(* IEC 61131-3 sources: tutorials/projects/ch05-2/PROGRAM, 4 files *)

(* ---- types.st ---- *)
(* 有初始化的数据类型 *)
TYPE BYTE_WITH_RANGE :
    SINT := 16#1A; (* 初始化为 0x1A *)
END_TYPE

(** 数组数据类型 *)
TYPE ARRAY_BYTES_WITH_RANGE :
    ARRAY [0..3] OF BYTE_WITH_RANGE;
END_TYPE

(* 枚举类型的数据类型: 机器状态 *)
TYPE ENUM_STATE_MACHINE : (
        INIT,
        PREPARING,
        RUNNING,
        STOPPED
    ) ;
END_TYPE

(*结构化的数据类型: 环境参数*)
TYPE STRUCT_ENV : STRUCT
        temperatures : ARRAY_BYTES_WITH_RANGE; (* 将多个温度值限制在10-60的范围 *)
        humity : REAL;
        state : ENUM_STATE_MACHINE;
    END_STRUCT ;
END_TYPE

(*嵌套结构化的数据类型*)
TYPE STRUCT_ENV_DATA :
    STRUCT
        env : STRUCT_ENV;
        dtime : TIME;
    END_STRUCT ;
END_TYPE

TYPE IOT_DATA :
    STRUCT_ENV_DATA;
END_TYPE

(* ---- funs.st ---- *)
FUNCTION func_sum_factorial : INT  (* 阶乘之和: 1!+2!+...+n! *)
    VAR_INPUT n: SINT; END_VAR

    VAR
        x: SINT;
        sum: INT := 0;
    END_VAR

    FOR x := 1 TO n DO
        sum := sum + func_factorial(x); (* 函数function调用function *)
    END_FOR;

    func_sum_factorial := sum;
END_FUNCTION

FUNCTION func_factorial : INT  (* n阶乘 !n 之和 *)
    VAR_INPUT n: SINT; END_VAR

    VAR
        x: SINT; sum: INT := 1;
    END_VAR

    FOR x := 1 TO n DO
        sum := sum*x;
    END_FOR;

    func_factorial := sum;
END_FUNCTION

FUNCTION func_sum_array : INT
    VAR_INPUT arrays: ARRAY_BYTES_WITH_RANGE; END_VAR
    VAR i: SINT; sum :INT :=0; END_VAR

    FOR i := 0 TO 3 BY 1 DO
        IF arrays[i] > 20 THEN
            sum := sum + 2;
        ELSE
            sum := sum + 1;
        END_IF;
    END_FOR;

    func_sum_array := sum;
END_FUNCTION

(* ---- fbs.st ---- *)
(* 功能块中可以调用其他功能块、函数 *)

FUNCTION_BLOCK fb_data_bank

        (* 功能块的输入: n, data*)
        VAR_INPUT
            n: INT; (*  *)
            data: STRUCT_ENV_DATA;
        END_VAR

        (* 功能块的输出: num, money*)
        VAR_OUTPUT
            money: DINT := 0;
            num: LINT := 0;
        END_VAR

        (* 功能块的功能逻辑: 将输入data中的数据累加到money中， 将输入n做阶乘累加到num中 *)
        money := money + func_sum_array(data.env.temperatures);
        num := func_factorial(n);

END_FUNCTION_BLOCK

(* ---- program-main.st ---- *)
(* PROGRAM 中可以调用其他POU， 如功能块、函数等 *)

PROGRAM program_demo_all_pous

    VAR
        (* 功能块使用前需要实例化 *)
        bank: fb_data_bank;
        (* 即将支持: 嵌套结构的初始化， 其中temperatures数组初始化为[20, 40, 40, 40] *)
        // iot_data: STRUCT_ENV_DATA := (dtime:=T#1d2h3m4s, env: (humity:=2.0, state:=RUNNING, temperatures:=[20,3(40)]));
        iot_data: STRUCT_ENV_DATA := (dtime:=T#4s);
        m_num: LINT := 0;
        money: DINT := 0;
    END_VAR

    (* 功能块调用时， 可以直接将某些输出赋值给变量：例如m_num *)
    bank(n := g_num, data := iot_data, num=>m_num);

    (* 功能块有数据记忆功能， 可以调用后将输出赋值给其他变量： 例如money *)
    money := bank.money;
    g_num := g_num + 1;

    (* 打印log时， 各个参数的类型需要与对应的占位符类型一致 *)
    WA_LOG('g_num=%d, m_num=%d, money=%d', g_num, m_num, money);

END_PROGRAM
